// TIA Portal V20 export
DATA_BLOCK "ManualOperationControl_U1Em2"   // DB207
// stored: MemoryReserve 100
   VAR
      manualOperationEm { ExternalAccessible := 'False'; ExternalVisible := 'False'; ExternalWritable := 'False'} : "LAF_typeManEm";
      manualOperationEmArea { ExternalAccessible := 'False'; ExternalVisible := 'False'; ExternalWritable := 'False'} : Array[1..2] of "LAF_typeManOperationArea";
      manualOperationCms { ExternalAccessible := 'False'; ExternalVisible := 'False'; ExternalWritable := 'False'} : Array[1..90] of "LAF_typeManOperation";
      axis { ExternalAccessible := 'False'; ExternalVisible := 'False'; ExternalWritable := 'False'} : Array[0..0] of "LBC_typeAxisControlInterface";
      axis64Pos { S7_SetPoint := 'True'} : Array[0..20] of "LBC_typeAxis64PosInterface";
      softCam { S7_SetPoint := 'True'} : Array[0..20] of "LER_typeSoftCamInterface2";
      twoWayActuator { S7_SetPoint := 'True'} : Array[0..14] of "LBC_typeTwoWayActuatorInterface";
   END_VAR
BEGIN
   manualOperationEm.equipmentModuleNum := 1030;
   manualOperationEm.actvArea := 0;
   manualOperationEm.pages.total := 0;
   manualOperationEm.pages.actv := 0;
   manualOperationEm.pages.numOfActvItems := 0;
   manualOperationEmArea[1..2].areaNum := 0;
   manualOperationEmArea[1].displayedLines := '1;';
   manualOperationEmArea[2].displayedLines := '21-33;';
   manualOperationEmArea[1..2].hmiPage.total := 0;
   manualOperationEmArea[1..2].hmiPage.actv := 0;
   manualOperationEmArea[1..2].hmiPage.numOfActvItems := 0;
   manualOperationCms[1..90].intf.lineNum := 0;
   manualOperationCms[1..90].intf.mode := 1;
   manualOperationCms[1..90].intf.showLine := FALSE;
   manualOperationCms[1..90].intf.enableMechAddr := FALSE;
   manualOperationCms[1..90].intf.expandable := FALSE;
   manualOperationCms[1..90].intf.disableLineSel := FALSE;
   manualOperationCms[1..90].intf.enableBigArea := FALSE;
   manualOperationCms[1..90].intf.cnfrmExecLeft := FALSE;
   manualOperationCms[1..90].intf.cnfrmExecRight := FALSE;
   manualOperationCms[1..90].intf.disableLeft := FALSE;
   manualOperationCms[1..90].intf.disableRight := FALSE;
   manualOperationCms[1..90].intf.cnfrmExecLeftCmd := FALSE;
   manualOperationCms[1..90].intf.cnfrmExecRightCmd := FALSE;
   manualOperationCms[1..90].intf.fieldDevAckLeft := FALSE;
   manualOperationCms[1..90].intf.fieldDevAckRight := FALSE;
   manualOperationCms[1..90].intf.nextLeftEndPos := 0;
   manualOperationCms[1..90].intf.nextRightEndPos := 0;
   manualOperationCms[1].intf.leftEndPosSens[0..7] := FALSE;
   manualOperationCms[2].intf.leftEndPosSens[0..7] := FALSE;
   manualOperationCms[3].intf.leftEndPosSens[0..7] := FALSE;
   manualOperationCms[4].intf.leftEndPosSens[0..7] := FALSE;
   manualOperationCms[5].intf.leftEndPosSens[0..7] := FALSE;
   manualOperationCms[6].intf.leftEndPosSens[0..7] := FALSE;
   manualOperationCms[7].intf.leftEndPosSens[0..7] := FALSE;
   manualOperationCms[8].intf.leftEndPosSens[0..7] := FALSE;
   manualOperationCms[9].intf.leftEndPosSens[0..7] := FALSE;
   manualOperationCms[10].intf.leftEndPosSens[0..7] := FALSE;
   manualOperationCms[11].intf.leftEndPosSens[0..7] := FALSE;
   manualOperationCms[12].intf.leftEndPosSens[0..7] := FALSE;
   manualOperationCms[13].intf.leftEndPosSens[0..7] := FALSE;
   manualOperationCms[14].intf.leftEndPosSens[0..7] := FALSE;
   manualOperationCms[15].intf.leftEndPosSens[0..7] := FALSE;
   manualOperationCms[16].intf.leftEndPosSens[0..7] := FALSE;
   manualOperationCms[17].intf.leftEndPosSens[0..7] := FALSE;
   manualOperationCms[18].intf.leftEndPosSens[0..7] := FALSE;
   manualOperationCms[19].intf.leftEndPosSens[0..7] := FALSE;
   manualOperationCms[20].intf.leftEndPosSens[0..7] := FALSE;
   manualOperationCms[21].intf.leftEndPosSens[0..7] := FALSE;
   manualOperationCms[22].intf.leftEndPosSens[0..7] := FALSE;
   manualOperationCms[23].intf.leftEndPosSens[0..7] := FALSE;
   manualOperationCms[24].intf.leftEndPosSens[0..7] := FALSE;
   manualOperationCms[25].intf.leftEndPosSens[0..7] := FALSE;
   manualOperationCms[26].intf.leftEndPosSens[0..7] := FALSE;
   manualOperationCms[27].intf.leftEndPosSens[0..7] := FALSE;
   manualOperationCms[28].intf.leftEndPosSens[0..7] := FALSE;
   manualOperationCms[29].intf.leftEndPosSens[0..7] := FALSE;
   manualOperationCms[30].intf.leftEndPosSens[0..7] := FALSE;
   manualOperationCms[31].intf.leftEndPosSens[0..7] := FALSE;
   manualOperationCms[32].intf.leftEndPosSens[0..7] := FALSE;
   manualOperationCms[33].intf.leftEndPosSens[0..7] := FALSE;
   manualOperationCms[34].intf.leftEndPosSens[0..7] := FALSE;
   manualOperationCms[35].intf.leftEndPosSens[0..7] := FALSE;
   manualOperationCms[36].intf.leftEndPosSens[0..7] := FALSE;
   manualOperationCms[37].intf.leftEndPosSens[0..7] := FALSE;
   manualOperationCms[38].intf.leftEndPosSens[0..7] := FALSE;
   manualOperationCms[39].intf.leftEndPosSens[0..7] := FALSE;
   manualOperationCms[40].intf.leftEndPosSens[0..7] := FALSE;
   manualOperationCms[41].intf.leftEndPosSens[0..7] := FALSE;
   manualOperationCms[42].intf.leftEndPosSens[0..7] := FALSE;
   manualOperationCms[43].intf.leftEndPosSens[0..7] := FALSE;
   manualOperationCms[44].intf.leftEndPosSens[0..7] := FALSE;
   manualOperationCms[45].intf.leftEndPosSens[0..7] := FALSE;
   manualOperationCms[46].intf.leftEndPosSens[0..7] := FALSE;
   manualOperationCms[47].intf.leftEndPosSens[0..7] := FALSE;
   manualOperationCms[48].intf.leftEndPosSens[0..7] := FALSE;
   manualOperationCms[49].intf.leftEndPosSens[0..7] := FALSE;
   manualOperationCms[50].intf.leftEndPosSens[0..7] := FALSE;
   manualOperationCms[51].intf.leftEndPosSens[0..7] := FALSE;
   manualOperationCms[52].intf.leftEndPosSens[0..7] := FALSE;
   manualOperationCms[53].intf.leftEndPosSens[0..7] := FALSE;
   manualOperationCms[54].intf.leftEndPosSens[0..7] := FALSE;
   manualOperationCms[55].intf.leftEndPosSens[0..7] := FALSE;
   manualOperationCms[56].intf.leftEndPosSens[0..7] := FALSE;
   manualOperationCms[57].intf.leftEndPosSens[0..7] := FALSE;
   manualOperationCms[58].intf.leftEndPosSens[0..7] := FALSE;
   manualOperationCms[59].intf.leftEndPosSens[0..7] := FALSE;
   manualOperationCms[60].intf.leftEndPosSens[0..7] := FALSE;
   manualOperationCms[61].intf.leftEndPosSens[0..7] := FALSE;
   manualOperationCms[62].intf.leftEndPosSens[0..7] := FALSE;
   manualOperationCms[63].intf.leftEndPosSens[0..7] := FALSE;
   manualOperationCms[64].intf.leftEndPosSens[0..7] := FALSE;
   manualOperationCms[65].intf.leftEndPosSens[0..7] := FALSE;
   manualOperationCms[66].intf.leftEndPosSens[0..7] := FALSE;
   manualOperationCms[67].intf.leftEndPosSens[0..7] := FALSE;
   manualOperationCms[68].intf.leftEndPosSens[0..7] := FALSE;
   manualOperationCms[69].intf.leftEndPosSens[0..7] := FALSE;
   manualOperationCms[70].intf.leftEndPosSens[0..7] := FALSE;
   manualOperationCms[71].intf.leftEndPosSens[0..7] := FALSE;
   manualOperationCms[72].intf.leftEndPosSens[0..7] := FALSE;
   manualOperationCms[73].intf.leftEndPosSens[0..7] := FALSE;
   manualOperationCms[74].intf.leftEndPosSens[0..7] := FALSE;
   manualOperationCms[75].intf.leftEndPosSens[0..7] := FALSE;
   manualOperationCms[76].intf.leftEndPosSens[0..7] := FALSE;
   manualOperationCms[77].intf.leftEndPosSens[0..7] := FALSE;
   manualOperationCms[78].intf.leftEndPosSens[0..7] := FALSE;
   manualOperationCms[79].intf.leftEndPosSens[0..7] := FALSE;
   manualOperationCms[80].intf.leftEndPosSens[0..7] := FALSE;
   manualOperationCms[81].intf.leftEndPosSens[0..7] := FALSE;
   manualOperationCms[82].intf.leftEndPosSens[0..7] := FALSE;
   manualOperationCms[83].intf.leftEndPosSens[0..7] := FALSE;
   manualOperationCms[84].intf.leftEndPosSens[0..7] := FALSE;
   manualOperationCms[85].intf.leftEndPosSens[0..7] := FALSE;
   manualOperationCms[86].intf.leftEndPosSens[0..7] := FALSE;
   manualOperationCms[87].intf.leftEndPosSens[0..7] := FALSE;
   manualOperationCms[88].intf.leftEndPosSens[0..7] := FALSE;
   manualOperationCms[89].intf.leftEndPosSens[0..7] := FALSE;
   manualOperationCms[90].intf.leftEndPosSens[0..7] := FALSE;
   manualOperationCms[1].intf.rightEndPosSens[0..7] := FALSE;
   manualOperationCms[2].intf.rightEndPosSens[0..7] := FALSE;
   manualOperationCms[3].intf.rightEndPosSens[0..7] := FALSE;
   manualOperationCms[4].intf.rightEndPosSens[0..7] := FALSE;
   manualOperationCms[5].intf.rightEndPosSens[0..7] := FALSE;
   manualOperationCms[6].intf.rightEndPosSens[0..7] := FALSE;
   manualOperationCms[7].intf.rightEndPosSens[0..7] := FALSE;
   manualOperationCms[8].intf.rightEndPosSens[0..7] := FALSE;
   manualOperationCms[9].intf.rightEndPosSens[0..7] := FALSE;
   manualOperationCms[10].intf.rightEndPosSens[0..7] := FALSE;
   manualOperationCms[11].intf.rightEndPosSens[0..7] := FALSE;
   manualOperationCms[12].intf.rightEndPosSens[0..7] := FALSE;
   manualOperationCms[13].intf.rightEndPosSens[0..7] := FALSE;
   manualOperationCms[14].intf.rightEndPosSens[0..7] := FALSE;
   manualOperationCms[15].intf.rightEndPosSens[0..7] := FALSE;
   manualOperationCms[16].intf.rightEndPosSens[0..7] := FALSE;
   manualOperationCms[17].intf.rightEndPosSens[0..7] := FALSE;
   manualOperationCms[18].intf.rightEndPosSens[0..7] := FALSE;
   manualOperationCms[19].intf.rightEndPosSens[0..7] := FALSE;
   manualOperationCms[20].intf.rightEndPosSens[0..7] := FALSE;
   manualOperationCms[21].intf.rightEndPosSens[0..7] := FALSE;
   manualOperationCms[22].intf.rightEndPosSens[0..7] := FALSE;
   manualOperationCms[23].intf.rightEndPosSens[0..7] := FALSE;
   manualOperationCms[24].intf.rightEndPosSens[0..7] := FALSE;
   manualOperationCms[25].intf.rightEndPosSens[0..7] := FALSE;
   manualOperationCms[26].intf.rightEndPosSens[0..7] := FALSE;
   manualOperationCms[27].intf.rightEndPosSens[0..7] := FALSE;
   manualOperationCms[28].intf.rightEndPosSens[0..7] := FALSE;
   manualOperationCms[29].intf.rightEndPosSens[0..7] := FALSE;
   manualOperationCms[30].intf.rightEndPosSens[0..7] := FALSE;
   manualOperationCms[31].intf.rightEndPosSens[0..7] := FALSE;
   manualOperationCms[32].intf.rightEndPosSens[0..7] := FALSE;
   manualOperationCms[33].intf.rightEndPosSens[0..7] := FALSE;
   manualOperationCms[34].intf.rightEndPosSens[0..7] := FALSE;
   manualOperationCms[35].intf.rightEndPosSens[0..7] := FALSE;
   manualOperationCms[36].intf.rightEndPosSens[0..7] := FALSE;
   manualOperationCms[37].intf.rightEndPosSens[0..7] := FALSE;
   manualOperationCms[38].intf.rightEndPosSens[0..7] := FALSE;
   manualOperationCms[39].intf.rightEndPosSens[0..7] := FALSE;
   manualOperationCms[40].intf.rightEndPosSens[0..7] := FALSE;
   manualOperationCms[41].intf.rightEndPosSens[0..7] := FALSE;
   manualOperationCms[42].intf.rightEndPosSens[0..7] := FALSE;
   manualOperationCms[43].intf.rightEndPosSens[0..7] := FALSE;
   manualOperationCms[44].intf.rightEndPosSens[0..7] := FALSE;
   manualOperationCms[45].intf.rightEndPosSens[0..7] := FALSE;
   manualOperationCms[46].intf.rightEndPosSens[0..7] := FALSE;
   manualOperationCms[47].intf.rightEndPosSens[0..7] := FALSE;
   manualOperationCms[48].intf.rightEndPosSens[0..7] := FALSE;
   manualOperationCms[49].intf.rightEndPosSens[0..7] := FALSE;
   manualOperationCms[50].intf.rightEndPosSens[0..7] := FALSE;
   manualOperationCms[51].intf.rightEndPosSens[0..7] := FALSE;
   manualOperationCms[52].intf.rightEndPosSens[0..7] := FALSE;
   manualOperationCms[53].intf.rightEndPosSens[0..7] := FALSE;
   manualOperationCms[54].intf.rightEndPosSens[0..7] := FALSE;
   manualOperationCms[55].intf.rightEndPosSens[0..7] := FALSE;
   manualOperationCms[56].intf.rightEndPosSens[0..7] := FALSE;
   manualOperationCms[57].intf.rightEndPosSens[0..7] := FALSE;
   manualOperationCms[58].intf.rightEndPosSens[0..7] := FALSE;
   manualOperationCms[59].intf.rightEndPosSens[0..7] := FALSE;
   manualOperationCms[60].intf.rightEndPosSens[0..7] := FALSE;
   manualOperationCms[61].intf.rightEndPosSens[0..7] := FALSE;
   manualOperationCms[62].intf.rightEndPosSens[0..7] := FALSE;
   manualOperationCms[63].intf.rightEndPosSens[0..7] := FALSE;
   manualOperationCms[64].intf.rightEndPosSens[0..7] := FALSE;
   manualOperationCms[65].intf.rightEndPosSens[0..7] := FALSE;
   manualOperationCms[66].intf.rightEndPosSens[0..7] := FALSE;
   manualOperationCms[67].intf.rightEndPosSens[0..7] := FALSE;
   manualOperationCms[68].intf.rightEndPosSens[0..7] := FALSE;
   manualOperationCms[69].intf.rightEndPosSens[0..7] := FALSE;
   manualOperationCms[70].intf.rightEndPosSens[0..7] := FALSE;
   manualOperationCms[71].intf.rightEndPosSens[0..7] := FALSE;
   manualOperationCms[72].intf.rightEndPosSens[0..7] := FALSE;
   manualOperationCms[73].intf.rightEndPosSens[0..7] := FALSE;
   manualOperationCms[74].intf.rightEndPosSens[0..7] := FALSE;
   manualOperationCms[75].intf.rightEndPosSens[0..7] := FALSE;
   manualOperationCms[76].intf.rightEndPosSens[0..7] := FALSE;
   manualOperationCms[77].intf.rightEndPosSens[0..7] := FALSE;
   manualOperationCms[78].intf.rightEndPosSens[0..7] := FALSE;
   manualOperationCms[79].intf.rightEndPosSens[0..7] := FALSE;
   manualOperationCms[80].intf.rightEndPosSens[0..7] := FALSE;
   manualOperationCms[81].intf.rightEndPosSens[0..7] := FALSE;
   manualOperationCms[82].intf.rightEndPosSens[0..7] := FALSE;
   manualOperationCms[83].intf.rightEndPosSens[0..7] := FALSE;
   manualOperationCms[84].intf.rightEndPosSens[0..7] := FALSE;
   manualOperationCms[85].intf.rightEndPosSens[0..7] := FALSE;
   manualOperationCms[86].intf.rightEndPosSens[0..7] := FALSE;
   manualOperationCms[87].intf.rightEndPosSens[0..7] := FALSE;
   manualOperationCms[88].intf.rightEndPosSens[0..7] := FALSE;
   manualOperationCms[89].intf.rightEndPosSens[0..7] := FALSE;
   manualOperationCms[90].intf.rightEndPosSens[0..7] := FALSE;
   manualOperationCms[1..90].intf.pos := 0.0;
   manualOperationCms[1..90].intf.minPos := 0.0;
   manualOperationCms[1..90].intf.maxPos := 0.0;
   manualOperationCms[1..90].intf.showPos := 0;
   manualOperationCms[1..90].cmd.lineSel := FALSE;
   manualOperationCms[1..90].cmd.expandedOemArea := FALSE;
   manualOperationCms[1..90].cmd.execLeftCmd := FALSE;
   manualOperationCms[1..90].cmd.execRightCmd := FALSE;
   manualOperationCms[1..90].cmd.disableLeftClick := FALSE;
   manualOperationCms[1..90].cmd.disableRightClick := FALSE;
   manualOperationCms[1..90].cmd.moreInfo := FALSE;
   manualOperationCms[1..90].cmd.actvAddr := 1;
   axis[0].commandConfiguration.generalSettings.stopOnError := TRUE;
   axis[0].commandConfiguration.generalSettings.resetWithRestart := FALSE;
   axis[0].commandConfiguration.generalSettings.abortWaitingSyncCmd := TRUE;
   axis[0].commandConfiguration.power.startMode := 1;
   axis[0].commandConfiguration.power.stopMode := 0;
   axis[0].commandConfiguration.power.syncMotionSimulation := FALSE;
   axis[0].commandConfiguration.power.syncMotionSimulationExtendedMode := -1;
   axis[0].commandConfiguration.jog.velocity := 0.0;
   axis[0].commandConfiguration.jog.acceleration := -1.0;
   axis[0].commandConfiguration.jog.deceleration := -1.0;
   axis[0].commandConfiguration.jog.jerk := -1.0;
   axis[0].commandConfiguration.jog.positionControlled := TRUE;
   axis[0].commandConfiguration.jog.increment := 0.0;
   axis[0].commandConfiguration.jog.mode := 0;
   axis[0].commandConfiguration.moveVelocity.velocity := 0.0;
   axis[0].commandConfiguration.moveVelocity.acceleration := -1.0;
   axis[0].commandConfiguration.moveVelocity.deceleration := -1.0;
   axis[0].commandConfiguration.moveVelocity.jerk := -1.0;
   axis[0].commandConfiguration.moveVelocity.direction := 0;
   axis[0].commandConfiguration.moveVelocity.positionControlled := TRUE;
   axis[0].commandConfiguration.moveVelocity.velocityChangeOnTheFly := FALSE;
   axis[0].commandConfiguration.stop.deceleration := -1.0;
   axis[0].commandConfiguration.stop.jerk := -1.0;
   axis[0].commandConfiguration.stop.abortAcceleration := FALSE;
   axis[0].commandConfiguration.fastStop.deceleration := -1.0;
   axis[0].commandConfiguration.fastStop.jerk := -1.0;
   axis[0].commandConfiguration.fastStop.abortAcceleration := FALSE;
   axis[0].commandConfiguration.fastStop.replaceStopPossible := FALSE;
   axis[0].commandConfiguration.torqueLimiting.limit := -1.0;
   axis[0].commandConfiguration.torqueLimiting.mode := 0;
   axis[0].commandConfiguration.homing.position := 0.0;
   axis[0].commandConfiguration.homing.mode := 0;
   axis[0].commandConfiguration.homing.sensor := 0;
   axis[0].commandConfiguration.homing.extendedMode := -1;
   axis[0].commandConfiguration.homing.extendedModeTorqueLimit := 0.0;
   axis[0].commandConfiguration.homing.extendedModeTargetPosition := 0.0;
   axis[0].commandConfiguration.posRelative.distance := 0.0;
   axis[0].commandConfiguration.posRelative.velocity := -1.0;
   axis[0].commandConfiguration.posRelative.acceleration := -1.0;
   axis[0].commandConfiguration.posRelative.deceleration := -1.0;
   axis[0].commandConfiguration.posRelative.jerk := -1.0;
   axis[0].commandConfiguration.posRelative.direction := 0;
   axis[0].commandConfiguration.posAbsolute.position := 0.0;
   axis[0].commandConfiguration.posAbsolute.velocity := -1.0;
   axis[0].commandConfiguration.posAbsolute.acceleration := -1.0;
   axis[0].commandConfiguration.posAbsolute.deceleration := -1.0;
   axis[0].commandConfiguration.posAbsolute.jerk := -1.0;
   axis[0].commandConfiguration.posAbsolute.direction := 1;
   axis[0].commandConfiguration.posAbsolute.positionChangeOnTheFly := FALSE;
   axis[0].commandConfiguration.posAbsolute.velocityChangeOnTheFly := FALSE;
   axis[0].commandConfiguration.posSuperimposed.distance := 0.0;
   axis[0].commandConfiguration.posSuperimposed.velocityDiff := -1.0;
   axis[0].commandConfiguration.posSuperimposed.acceleration := -1.0;
   axis[0].commandConfiguration.posSuperimposed.deceleration := -1.0;
   axis[0].commandConfiguration.posSuperimposed.jerk := -1.0;
   axis[0].commandConfiguration.posSuperimposed.direction := 0;
   axis[0].commandConfiguration.haltSuperimposed.deceleration := -1.0;
   axis[0].commandConfiguration.haltSuperimposed.jerk := -1.0;
   axis[0].commandConfiguration.haltSuperimposed.abortAcceleration := FALSE;
   axis[0].commandConfiguration.gearInRelative.ratioNumerator := 1;
   axis[0].commandConfiguration.gearInRelative.ratioDenominator := 1;
   axis[0].commandConfiguration.gearInRelative.acceleration := -1.0;
   axis[0].commandConfiguration.gearInRelative.deceleration := -1.0;
   axis[0].commandConfiguration.gearInRelative.jerk := -1.0;
   axis[0].commandConfiguration.gearInRelative.ratioChangeOnTheFly := FALSE;
   axis[0].commandConfiguration.gearInAbsolute.ratioNumerator := 1;
   axis[0].commandConfiguration.gearInAbsolute.ratioDenominator := 1;
   axis[0].commandConfiguration.gearInAbsolute.masterSyncPosition := 0.0;
   axis[0].commandConfiguration.gearInAbsolute.slaveSyncPosition := 0.0;
   axis[0].commandConfiguration.gearInAbsolute.syncProfileReference := 1;
   axis[0].commandConfiguration.gearInAbsolute.masterStartDistance := 0.0;
   axis[0].commandConfiguration.gearInAbsolute.velocity := -1.0;
   axis[0].commandConfiguration.gearInAbsolute.acceleration := -1.0;
   axis[0].commandConfiguration.gearInAbsolute.deceleration := -1.0;
   axis[0].commandConfiguration.gearInAbsolute.jerk := -1.0;
   axis[0].commandConfiguration.gearInAbsolute.syncDirection := 1;
   axis[0].commandConfiguration.gearInAbsolute.ratioChangeOnTheFly := FALSE;
   axis[0].commandConfiguration.gearInVelocity.continuousUpdate := FALSE;
   axis[0].commandConfiguration.gearInVelocity.ratioNumerator := 1;
   axis[0].commandConfiguration.gearInVelocity.ratioDenominator := 1;
   axis[0].commandConfiguration.gearInVelocity.acceleration := -1.0;
   axis[0].commandConfiguration.gearInVelocity.deceleration := -1.0;
   axis[0].commandConfiguration.gearInVelocity.jerk := -1.0;
   axis[0].commandConfiguration.gearInVelocity.positionControlled := FALSE;
   axis[0].commandConfiguration.camIn.masterOffset := 0.0;
   axis[0].commandConfiguration.camIn.slaveOffset := 0.0;
   axis[0].commandConfiguration.camIn.masterScaling := 1.0;
   axis[0].commandConfiguration.camIn.slaveScaling := 1.0;
   axis[0].commandConfiguration.camIn.masterSyncPosition := 0.0;
   axis[0].commandConfiguration.camIn.syncProfileReference := 1;
   axis[0].commandConfiguration.camIn.masterStartDistance := 0.0;
   axis[0].commandConfiguration.camIn.velocity := -1.0;
   axis[0].commandConfiguration.camIn.acceleration := -1.0;
   axis[0].commandConfiguration.camIn.deceleration := -1.0;
   axis[0].commandConfiguration.camIn.jerk := -1.0;
   axis[0].commandConfiguration.camIn.applicationMode := 0;
   axis[0].commandConfiguration.camIn.syncDirection := 1;
   axis[0].commandConfiguration.gearOutCamOut.slavePosition := 0.0;
   axis[0].commandConfiguration.gearOutCamOut.syncProfileReference := 1;
   axis[0].commandConfiguration.gearOutCamOut.masterStopDistance := 0.0;
   axis[0].commandConfiguration.gearOutCamOut.deceleration := -1.0;
   axis[0].commandConfiguration.gearOutCamOut.jerk := -1.0;
   axis[0].commandConfiguration.gearOutCamOut.syncOutDirection := 3;
   axis[0].commandConfiguration.gearOutCamOut.gearOutCamOutMode := -1;
   axis[0].commandConfiguration.phasing.phaseShift := 0.0;
   axis[0].commandConfiguration.phasing.velocity := -1.0;
   axis[0].commandConfiguration.phasing.acceleration := -1.0;
   axis[0].commandConfiguration.phasing.deceleration := -1.0;
   axis[0].commandConfiguration.phasing.jerk := -1.0;
   axis[0].commandConfiguration.phasing.profileReference := 0;
   axis[0].commandConfiguration.phasing.phasingDistance := 0.0;
   axis[0].commandConfiguration.phasing.startPosition := 0.0;
   axis[0].commandConfiguration.phasing.direction := 3;
   axis[0].commandConfiguration.phasing.phaseAbsolute := TRUE;
   axis[0].commandConfiguration.phasing.phaseShiftChangeOnTheFly := FALSE;
   axis[0].commandConfiguration.offset.offset := 0.0;
   axis[0].commandConfiguration.offset.profileReference := 1;
   axis[0].commandConfiguration.offset.offsetDistance := 0.0;
   axis[0].commandConfiguration.offset.startPosition := 0.0;
   axis[0].commandConfiguration.offset.direction := 3;
   axis[0].commandConfiguration.offset.offsetAbsolute := TRUE;
   axis[0].commandConfiguration.offset.offsetChangeOnTheFly := FALSE;
   axis[0].commands.enable := FALSE;
   axis[0].commands.enableAxis := FALSE;
   axis[0].commands.resetAxis := FALSE;
   axis[0].commands.openBrake := FALSE;
   axis[0].commands.jogForward := FALSE;
   axis[0].commands.jogBackward := FALSE;
   axis[0].commands.moveVelocity := FALSE;
   axis[0].commands.stop := FALSE;
   axis[0].commands.fastStop := FALSE;
   axis[0].commands.torqueLimiting := FALSE;
   axis[0].commands.homing := FALSE;
   axis[0].commands.posRelative := FALSE;
   axis[0].commands.posAbsolute := FALSE;
   axis[0].commands.posSuperimposed := FALSE;
   axis[0].commands.haltSuperimposed := FALSE;
   axis[0].commands.gearInRelative := FALSE;
   axis[0].commands.gearInAbsolute := FALSE;
   axis[0].commands.gearInVelocity := FALSE;
   axis[0].commands.camIn := FALSE;
   axis[0].commands.gearOutCamOut := FALSE;
   axis[0].commands.phasing := FALSE;
   axis[0].commands.offset := FALSE;
   axis[0].commands.refreshConfiguration := FALSE;
   axis[0].commands.editConfiguration := FALSE;
   axis[0].commands.saveConfiguration := FALSE;
   axis[0].commands.uploadCurrentTorque := FALSE;
   axis[0].commands.reset := FALSE;
   axis[0].monitoring.enable := FALSE;
   axis[0].monitoring.referenceDesignator := WSTRING#'';
   axis[0].monitoring.enabled := FALSE;
   axis[0].monitoring.resetAxis := FALSE;
   axis[0].monitoring.moveVelocity := FALSE;
   axis[0].monitoring.fastStop := FALSE;
   axis[0].monitoring.stop := FALSE;
   axis[0].monitoring.homing := FALSE;
   axis[0].monitoring.posRelative := FALSE;
   axis[0].monitoring.posAbsolute := FALSE;
   axis[0].monitoring.posSuperimposed := FALSE;
   axis[0].monitoring.haltSuperimposed := FALSE;
   axis[0].monitoring.gearInRelative := FALSE;
   axis[0].monitoring.offset := FALSE;
   axis[0].monitoring.phasing := FALSE;
   axis[0].monitoring.gearOutCamOut := FALSE;
   axis[0].monitoring.camIn := FALSE;
   axis[0].monitoring.gearInVelocity := FALSE;
   axis[0].monitoring.gearInAbsolute := FALSE;
   axis[0].monitoring.reset := FALSE;
   axis[0].monitoring.enableAxis := FALSE;
   axis[0].monitoring.openBrake := FALSE;
   axis[0].monitoring.torqueLimiting := FALSE;
   axis[0].monitoring.enableManualCmds := FALSE;
   axis[0].monitoring.jogBackward := FALSE;
   axis[0].monitoring.jogForward := FALSE;
   axis[0].monitoring.brakeOpened := FALSE;
   axis[0].monitoring.axisEnabled := FALSE;
   axis[0].monitoring.resetActive := FALSE;
   axis[0].monitoring.inVelocity := FALSE;
   axis[0].monitoring.inLimitation := FALSE;
   axis[0].monitoring.inClamping := FALSE;
   axis[0].monitoring.startSync := FALSE;
   axis[0].monitoring.inSync := FALSE;
   axis[0].monitoring.inSimulation := FALSE;
   axis[0].monitoring.jogSelected := FALSE;
   axis[0].monitoring.moveVelocitySelected := FALSE;
   axis[0].monitoring.stopSelected := FALSE;
   axis[0].monitoring.fastStopSelected := FALSE;
   axis[0].monitoring.torqueLimitingSelected := FALSE;
   axis[0].monitoring.homingSelected := FALSE;
   axis[0].monitoring.posRelativeSelected := FALSE;
   axis[0].monitoring.posAbsoluteSelected := FALSE;
   axis[0].monitoring.posSuperimposedSelected := FALSE;
   axis[0].monitoring.haltSuperimposedSelected := FALSE;
   axis[0].monitoring.gearInRelativeSelected := FALSE;
   axis[0].monitoring.gearInAbsoluteSelected := FALSE;
   axis[0].monitoring.gearInVelocitySelected := FALSE;
   axis[0].monitoring.camInSelected := FALSE;
   axis[0].monitoring.gearOutCamOutSelected := FALSE;
   axis[0].monitoring.phasingSelected := FALSE;
   axis[0].monitoring.offsetSelected := FALSE;
   axis[0].monitoring.commandBusy := FALSE;
   axis[0].monitoring.commandDone := FALSE;
   axis[0].monitoring.commandAborted := FALSE;
   axis[0].monitoring.homingCommandBusy := FALSE;
   axis[0].monitoring.homingCommandDone := FALSE;
   axis[0].monitoring.homingCommandAborted := FALSE;
   axis[0].monitoring.superimposedBusy := FALSE;
   axis[0].monitoring.superimposedDone := FALSE;
   axis[0].monitoring.superimposedAborted := FALSE;
   axis[0].monitoring.interlockGeneral := FALSE;
   axis[0].monitoring.interlockJogForward := FALSE;
   axis[0].monitoring.interlockJogBackward := FALSE;
   axis[0].monitoring.interlockWarningGeneral := FALSE;
   axis[0].monitoring.interlockWarningJogForward := FALSE;
   axis[0].monitoring.interlockWarningJogBackward := FALSE;
   axis[0].monitoring.valid := FALSE;
   axis[0].monitoring.busy := FALSE;
   axis[0].monitoring.error := FALSE;
   axis[0].monitoring.status := 16#0000;
   axis[0].monitoring.subfunctionStatus := 16#0000;
   axis[0].monitoring.actualPosition := 0.0;
   axis[0].monitoring.actualSpeed := 0.0;
   axis[0].monitoring.speedUnit := 0;
   axis[0].monitoring.positionUnit := 0;
   axis[0].monitoring.axisStatus1 := 16#0000_0000;
   axis[0].monitoring.axisStatus2 := 16#0000_0000;
   axis[0].monitoring.axisType := 0;
   axis[0].monitoring.maxVelocity := 0.0;
   axis[0].monitoring.actualCurrent := 0.0;
   axis[0].monitoring.actualTorque := 0.0;
   axis[0].monitoring.velocityOverrideEnabled := FALSE;
   axis[0].monitoring.sinaParaError := FALSE;
   axis[0].monitoring.sinaParaStatus := 16#0000_0000;
   axis[0].configuration.referenceDesignator := WSTRING#'AxisControl';
   axis[0].configuration.disableAlarms := FALSE;
   axis[0].configuration.masterControlPopUp := TRUE;
   axis64Pos[0].commandConfiguration.generalSettings.stopOnError := TRUE;
   axis64Pos[0].commandConfiguration.generalSettings.resetWithRestart := FALSE;
   axis64Pos[0].commandConfiguration.generalSettings.abortWaitingSyncCmd := TRUE;
   axis64Pos[0].commandConfiguration.power.startMode := 1;
   axis64Pos[0].commandConfiguration.power.stopMode := 0;
   axis64Pos[0].commandConfiguration.power.syncMotionSimulation := FALSE;
   axis64Pos[0].commandConfiguration.power.syncMotionSimulationExtendedMode := -1;
   axis64Pos[0].commandConfiguration.jog.velocity := 0.0;
   axis64Pos[0].commandConfiguration.jog.acceleration := -1.0;
   axis64Pos[0].commandConfiguration.jog.deceleration := -1.0;
   axis64Pos[0].commandConfiguration.jog.jerk := -1.0;
   axis64Pos[0].commandConfiguration.jog.positionControlled := TRUE;
   axis64Pos[0].commandConfiguration.jog.increment := 0.0;
   axis64Pos[0].commandConfiguration.jog.mode := 0;
   axis64Pos[0].commandConfiguration.moveVelocity.velocity := 0.0;
   axis64Pos[0].commandConfiguration.moveVelocity.acceleration := -1.0;
   axis64Pos[0].commandConfiguration.moveVelocity.deceleration := -1.0;
   axis64Pos[0].commandConfiguration.moveVelocity.jerk := -1.0;
   axis64Pos[0].commandConfiguration.moveVelocity.direction := 0;
   axis64Pos[0].commandConfiguration.moveVelocity.positionControlled := TRUE;
   axis64Pos[0].commandConfiguration.moveVelocity.velocityChangeOnTheFly := FALSE;
   axis64Pos[0].commandConfiguration.stop.deceleration := -1.0;
   axis64Pos[0].commandConfiguration.stop.jerk := -1.0;
   axis64Pos[0].commandConfiguration.stop.abortAcceleration := FALSE;
   axis64Pos[0].commandConfiguration.fastStop.deceleration := -1.0;
   axis64Pos[0].commandConfiguration.fastStop.jerk := -1.0;
   axis64Pos[0].commandConfiguration.fastStop.abortAcceleration := FALSE;
   axis64Pos[0].commandConfiguration.fastStop.replaceStopPossible := FALSE;
   axis64Pos[0].commandConfiguration.torqueLimiting.limit := -1.0;
   axis64Pos[0].commandConfiguration.torqueLimiting.mode := 0;
   axis64Pos[0].commandConfiguration.homing.position := 0.0;
   axis64Pos[0].commandConfiguration.homing.mode := 0;
   axis64Pos[0].commandConfiguration.homing.sensor := 0;
   axis64Pos[0].commandConfiguration.homing.extendedMode := -1;
   axis64Pos[0].commandConfiguration.homing.extendedModeTorqueLimit := 0.0;
   axis64Pos[0].commandConfiguration.homing.extendedModeTargetPosition := 0.0;
   axis64Pos[0].commandConfiguration.posRelative.distance := 0.0;
   axis64Pos[0].commandConfiguration.posRelative.velocity := -1.0;
   axis64Pos[0].commandConfiguration.posRelative.acceleration := -1.0;
   axis64Pos[0].commandConfiguration.posRelative.deceleration := -1.0;
   axis64Pos[0].commandConfiguration.posRelative.jerk := -1.0;
   axis64Pos[0].commandConfiguration.posRelative.direction := 0;
   axis64Pos[0].commandConfiguration.posAbsolute.position := 0.0;
   axis64Pos[0].commandConfiguration.posAbsolute.velocity := -1.0;
   axis64Pos[0].commandConfiguration.posAbsolute.acceleration := -1.0;
   axis64Pos[0].commandConfiguration.posAbsolute.deceleration := -1.0;
   axis64Pos[0].commandConfiguration.posAbsolute.jerk := -1.0;
   axis64Pos[0].commandConfiguration.posAbsolute.direction := 1;
   axis64Pos[0].commandConfiguration.posAbsolute.positionChangeOnTheFly := FALSE;
   axis64Pos[0].commandConfiguration.posAbsolute.velocityChangeOnTheFly := FALSE;
   axis64Pos[0].commandConfiguration.posSuperimposed.distance := 0.0;
   axis64Pos[0].commandConfiguration.posSuperimposed.velocityDiff := -1.0;
   axis64Pos[0].commandConfiguration.posSuperimposed.acceleration := -1.0;
   axis64Pos[0].commandConfiguration.posSuperimposed.deceleration := -1.0;
   axis64Pos[0].commandConfiguration.posSuperimposed.jerk := -1.0;
   axis64Pos[0].commandConfiguration.posSuperimposed.direction := 0;
   axis64Pos[0].commandConfiguration.haltSuperimposed.deceleration := -1.0;
   axis64Pos[0].commandConfiguration.haltSuperimposed.jerk := -1.0;
   axis64Pos[0].commandConfiguration.haltSuperimposed.abortAcceleration := FALSE;
   axis64Pos[0].commandConfiguration.gearInRelative.ratioNumerator := 1;
   axis64Pos[0].commandConfiguration.gearInRelative.ratioDenominator := 1;
   axis64Pos[0].commandConfiguration.gearInRelative.acceleration := -1.0;
   axis64Pos[0].commandConfiguration.gearInRelative.deceleration := -1.0;
   axis64Pos[0].commandConfiguration.gearInRelative.jerk := -1.0;
   axis64Pos[0].commandConfiguration.gearInRelative.ratioChangeOnTheFly := FALSE;
   axis64Pos[0].commandConfiguration.gearInAbsolute.ratioNumerator := 1;
   axis64Pos[0].commandConfiguration.gearInAbsolute.ratioDenominator := 1;
   axis64Pos[0].commandConfiguration.gearInAbsolute.masterSyncPosition := 0.0;
   axis64Pos[0].commandConfiguration.gearInAbsolute.slaveSyncPosition := 0.0;
   axis64Pos[0].commandConfiguration.gearInAbsolute.syncProfileReference := 1;
   axis64Pos[0].commandConfiguration.gearInAbsolute.masterStartDistance := 0.0;
   axis64Pos[0].commandConfiguration.gearInAbsolute.velocity := -1.0;
   axis64Pos[0].commandConfiguration.gearInAbsolute.acceleration := -1.0;
   axis64Pos[0].commandConfiguration.gearInAbsolute.deceleration := -1.0;
   axis64Pos[0].commandConfiguration.gearInAbsolute.jerk := -1.0;
   axis64Pos[0].commandConfiguration.gearInAbsolute.syncDirection := 1;
   axis64Pos[0].commandConfiguration.gearInAbsolute.ratioChangeOnTheFly := FALSE;
   axis64Pos[0].commandConfiguration.gearInVelocity.continuousUpdate := FALSE;
   axis64Pos[0].commandConfiguration.gearInVelocity.ratioNumerator := 1;
   axis64Pos[0].commandConfiguration.gearInVelocity.ratioDenominator := 1;
   axis64Pos[0].commandConfiguration.gearInVelocity.acceleration := -1.0;
   axis64Pos[0].commandConfiguration.gearInVelocity.deceleration := -1.0;
   axis64Pos[0].commandConfiguration.gearInVelocity.jerk := -1.0;
   axis64Pos[0].commandConfiguration.gearInVelocity.positionControlled := FALSE;
   axis64Pos[0].commandConfiguration.camIn.masterOffset := 0.0;
   axis64Pos[0].commandConfiguration.camIn.slaveOffset := 0.0;
   axis64Pos[0].commandConfiguration.camIn.masterScaling := 1.0;
   axis64Pos[0].commandConfiguration.camIn.slaveScaling := 1.0;
   axis64Pos[0].commandConfiguration.camIn.masterSyncPosition := 0.0;
   axis64Pos[0].commandConfiguration.camIn.syncProfileReference := 1;
   axis64Pos[0].commandConfiguration.camIn.masterStartDistance := 0.0;
   axis64Pos[0].commandConfiguration.camIn.velocity := -1.0;
   axis64Pos[0].commandConfiguration.camIn.acceleration := -1.0;
   axis64Pos[0].commandConfiguration.camIn.deceleration := -1.0;
   axis64Pos[0].commandConfiguration.camIn.jerk := -1.0;
   axis64Pos[0].commandConfiguration.camIn.applicationMode := 0;
   axis64Pos[0].commandConfiguration.camIn.syncDirection := 1;
   axis64Pos[0].commandConfiguration.gearOutCamOut.slavePosition := 0.0;
   axis64Pos[0].commandConfiguration.gearOutCamOut.syncProfileReference := 1;
   axis64Pos[0].commandConfiguration.gearOutCamOut.masterStopDistance := 0.0;
   axis64Pos[0].commandConfiguration.gearOutCamOut.deceleration := -1.0;
   axis64Pos[0].commandConfiguration.gearOutCamOut.jerk := -1.0;
   axis64Pos[0].commandConfiguration.gearOutCamOut.syncOutDirection := 3;
   axis64Pos[0].commandConfiguration.gearOutCamOut.gearOutCamOutMode := -1;
   axis64Pos[0].commandConfiguration.phasing.phaseShift := 0.0;
   axis64Pos[0].commandConfiguration.phasing.velocity := -1.0;
   axis64Pos[0].commandConfiguration.phasing.acceleration := -1.0;
   axis64Pos[0].commandConfiguration.phasing.deceleration := -1.0;
   axis64Pos[0].commandConfiguration.phasing.jerk := -1.0;
   axis64Pos[0].commandConfiguration.phasing.profileReference := 0;
   axis64Pos[0].commandConfiguration.phasing.phasingDistance := 0.0;
   axis64Pos[0].commandConfiguration.phasing.startPosition := 0.0;
   axis64Pos[0].commandConfiguration.phasing.direction := 3;
   axis64Pos[0].commandConfiguration.phasing.phaseAbsolute := TRUE;
   axis64Pos[0].commandConfiguration.phasing.phaseShiftChangeOnTheFly := FALSE;
   axis64Pos[0].commandConfiguration.offset.offset := 0.0;
   axis64Pos[0].commandConfiguration.offset.profileReference := 1;
   axis64Pos[0].commandConfiguration.offset.offsetDistance := 0.0;
   axis64Pos[0].commandConfiguration.offset.startPosition := 0.0;
   axis64Pos[0].commandConfiguration.offset.direction := 3;
   axis64Pos[0].commandConfiguration.offset.offsetAbsolute := TRUE;
   axis64Pos[0].commandConfiguration.offset.offsetChangeOnTheFly := FALSE;
   axis64Pos[0].commands.enableMasterControl := FALSE;
   axis64Pos[0].commands.enableAxis := FALSE;
   axis64Pos[0].commands.resetAxis := FALSE;
   axis64Pos[0].commands.openBrake := FALSE;
   axis64Pos[0].commands.jogForward := FALSE;
   axis64Pos[0].commands.jogBackward := FALSE;
   axis64Pos[0].commands.moveVelocity := FALSE;
   axis64Pos[0].commands.stop := FALSE;
   axis64Pos[0].commands.fastStop := FALSE;
   axis64Pos[0].commands.torqueLimiting := FALSE;
   axis64Pos[0].commands.homing := FALSE;
   axis64Pos[0].commands.posRelative := FALSE;
   axis64Pos[0].commands.posAbsolute := FALSE;
   axis64Pos[0].commands.posSuperimposed := FALSE;
   axis64Pos[0].commands.haltSuperimposed := FALSE;
   axis64Pos[0].commands.selectSetPosition := 0;
   axis64Pos[0].commands.uploadParameters := FALSE;
   axis64Pos[0].commands.refreshConfiguration := FALSE;
   axis64Pos[0].commands.editConfiguration := FALSE;
   axis64Pos[0].commands.saveConfiguration := FALSE;
   axis64Pos[0].commands.uploadCurrentTorque := FALSE;
   axis64Pos[0].commands.reset := FALSE;
   axis64Pos[0].monitoring.enable := FALSE;
   axis64Pos[0].monitoring.referenceDesignator := WSTRING#'';
   axis64Pos[0].monitoring.enabled := FALSE;
   axis64Pos[0].monitoring.enableManualCmds := FALSE;
   axis64Pos[0].monitoring.reset := FALSE;
   axis64Pos[0].monitoring.resetAxis := FALSE;
   axis64Pos[0].monitoring.enableAxis := FALSE;
   axis64Pos[0].monitoring.openBrake := FALSE;
   axis64Pos[0].monitoring.jogBackward := FALSE;
   axis64Pos[0].monitoring.jogForward := FALSE;
   axis64Pos[0].monitoring.moveVelocity := FALSE;
   axis64Pos[0].monitoring.stop := FALSE;
   axis64Pos[0].monitoring.fastStop := FALSE;
   axis64Pos[0].monitoring.torqueLimiting := FALSE;
   axis64Pos[0].monitoring.homing := FALSE;
   axis64Pos[0].monitoring.posRelative := FALSE;
   axis64Pos[0].monitoring.posAbsolute := FALSE;
   axis64Pos[0].monitoring.posSuperimposed := FALSE;
   axis64Pos[0].monitoring.haltSuperimposed := FALSE;
   axis64Pos[0].monitoring.brakeOpened := FALSE;
   axis64Pos[0].monitoring.axisEnabled := FALSE;
   axis64Pos[0].monitoring.resetActive := FALSE;
   axis64Pos[0].monitoring.inVelocity := FALSE;
   axis64Pos[0].monitoring.inLimitation := FALSE;
   axis64Pos[0].monitoring.inClamping := FALSE;
   axis64Pos[0].monitoring.startSync := FALSE;
   axis64Pos[0].monitoring.inSync := FALSE;
   axis64Pos[0].monitoring.inSimulation := FALSE;
   axis64Pos[0].monitoring.jogSelected := FALSE;
   axis64Pos[0].monitoring.moveVelocitySelected := FALSE;
   axis64Pos[0].monitoring.stopSelected := FALSE;
   axis64Pos[0].monitoring.fastStopSelected := FALSE;
   axis64Pos[0].monitoring.torqueLimitingSelected := FALSE;
   axis64Pos[0].monitoring.homingSelected := FALSE;
   axis64Pos[0].monitoring.posRelativeSelected := FALSE;
   axis64Pos[0].monitoring.posAbsoluteSelected := FALSE;
   axis64Pos[0].monitoring.posSuperimposedSelected := FALSE;
   axis64Pos[0].monitoring.haltSuperimposedSelected := FALSE;
   axis64Pos[0].monitoring.commandBusy := FALSE;
   axis64Pos[0].monitoring.commandDone := FALSE;
   axis64Pos[0].monitoring.commandAborted := FALSE;
   axis64Pos[0].monitoring.homingCommandBusy := FALSE;
   axis64Pos[0].monitoring.homingCommandDone := FALSE;
   axis64Pos[0].monitoring.homingCommandAborted := FALSE;
   axis64Pos[0].monitoring.superimposedBusy := FALSE;
   axis64Pos[0].monitoring.superimposedDone := FALSE;
   axis64Pos[0].monitoring.superimposedAborted := FALSE;
   axis64Pos[0].monitoring.selectSetPosition := 0;
   axis64Pos[0].monitoring.selectionController := TRUE;
   axis64Pos[0].monitoring.interlockGeneral := FALSE;
   axis64Pos[0].monitoring.interlockJogForward := FALSE;
   axis64Pos[0].monitoring.interlockJogBackward := FALSE;
   axis64Pos[0].monitoring.interlockWarningGeneral := FALSE;
   axis64Pos[0].monitoring.interlockWarningJogForward := FALSE;
   axis64Pos[0].monitoring.interlockWarningJogBackward := FALSE;
   axis64Pos[0].monitoring.valid := FALSE;
   axis64Pos[0].monitoring.busy := FALSE;
   axis64Pos[0].monitoring.error := FALSE;
   axis64Pos[0].monitoring.status := 16#0000;
   axis64Pos[0].monitoring.subfunctionStatus := 16#0000;
   axis64Pos[0].monitoring.actualPosition := 0.0;
   axis64Pos[0].monitoring.actualSpeed := 0.0;
   axis64Pos[0].monitoring.speedUnit := 0;
   axis64Pos[0].monitoring.positionUnit := 0;
   axis64Pos[0].monitoring.axisType := 0;
   axis64Pos[0].monitoring.maxVelocity := 0.0;
   axis64Pos[0].monitoring.actualCurrent := 0.0;
   axis64Pos[0].monitoring.actualTorque := 0.0;
   axis64Pos[0].monitoring.velocityOverrideEnabled := FALSE;
   axis64Pos[0].monitoring.sinaParaError := FALSE;
   axis64Pos[0].monitoring.sinaParaStatus := 16#0000_0000;
   axis64Pos[0].configuration.referenceDesignator := WSTRING#'Axis64Pos';
   axis64Pos[0].configuration.disableAlarms := FALSE;
   axis64Pos[0].configuration.masterControlPopUp := TRUE;
   axis64Pos[0].configuration.setPositions[0..15].position := 0.0;
   axis64Pos[0].configuration.setPositions[0..15].velocity := -1.0;
   axis64Pos[0].configuration.setPositions[0..15].acceleration := -1.0;
   axis64Pos[0].configuration.setPositions[0..15].deceleration := -1.0;
   axis64Pos[0].configuration.setPositions[0..15]."name" := '';
   twoWayActuator[0..13].commands.refreshConfiguration := FALSE;
   twoWayActuator[0..13].commands.editConfiguration := FALSE;
   twoWayActuator[0..13].commands.saveConfiguration := FALSE;
   twoWayActuator[0..13].commands.reset := FALSE;
   twoWayActuator[0..13].commands.commandHomePos := FALSE;
   twoWayActuator[0..13].commands.commandWorkPos := FALSE;
   twoWayActuator[0..13].monitoring.enable := FALSE;
   twoWayActuator[0..13].monitoring.referenceDesignator := WSTRING#'';
   twoWayActuator[0..13].monitoring.commandHomePos := FALSE;
   twoWayActuator[0..13].monitoring.commandWorkPos := FALSE;
   twoWayActuator[0..13].monitoring.goToHomePos := FALSE;
   twoWayActuator[0..13].monitoring.goToWorkPos := FALSE;
   twoWayActuator[0..13].monitoring.inHomePos := FALSE;
   twoWayActuator[0..13].monitoring.inWorkPos := FALSE;
   twoWayActuator[0..13].monitoring.reset := FALSE;
   twoWayActuator[0..13].monitoring.enableManualCmds := FALSE;
   twoWayActuator[0..13].monitoring.error := FALSE;
   twoWayActuator[0..13].monitoring.interlockHomePos := FALSE;
   twoWayActuator[0..13].monitoring.interlockWorkPos := FALSE;
   twoWayActuator[0..13].monitoring.status := 16#0000;
   twoWayActuator[0..13].monitoring.interlockWarningWorkPos := FALSE;
   twoWayActuator[0..13].monitoring.interlockWarningHomePos := FALSE;
   twoWayActuator[0..13].configuration.referenceDesignator := WSTRING#'TwoWayAct.';
   twoWayActuator[0..13].configuration.monitoringLeavingFeedback := T#5S;
   twoWayActuator[0..13].configuration.monitoringReachingFeedback := T#5S;
   twoWayActuator[0..13].configuration.monitoringDiscrepancy := T#0MS;
   twoWayActuator[0..13].configuration.setOutputHomeContinuously := TRUE;
   twoWayActuator[0..13].configuration.setOutputWorkContinuously := TRUE;
   twoWayActuator[0..13].configuration.disableHomeCommand := FALSE;
   twoWayActuator[0..13].configuration.disableFeedbackHomePos := FALSE;
   twoWayActuator[0..13].configuration.disableFeedbackWorkPos := FALSE;
   twoWayActuator[0..13].configuration.disableAlarms := FALSE;
   twoWayActuator[0..13].configuration.resetOutputsOnError := FALSE;
   twoWayActuator[0..13].configuration.allwaysWaitOnReachingTime := FALSE;
END_DATA_BLOCK
